FUNCTION_BLOCK FB_PackML_ExternalControl IMPLEMENTS ITF_PackML_ExternalControl
VAR_INPUT
END_VAR
VAR_OUTPUT
END_VAR
VAR
	nMode				: DINT;
	nModeCommand		: DINT;
	bModeCommandPulse	: BOOL;
	eState				: Tc3_PackML_V2.E_PMLState;
	eStateCommand		: Tc3_PackML_V2.E_PMLCommand;
	bStateCommandPulse	: BOOL;
	
	bStartPressed		: BOOL;
	bStartEnabled		: BOOL;
	bStopPressed		: BOOL;
	bStopEnabled		: BOOL;
	bResetPressed		: BOOL;
	bResetEnabled		: BOOL;
	bClearPressed		: BOOL;
	bClearEnabled		: BOOL;	
	
END_VAR

//Handle button presses
IF bStartPressed THEN
	IF eState = Tc3_PackML_V2.E_PMLState.ePMLState_Idle THEN
		eStateCommand := Tc3_PackML_V2.E_PMLCommand.ePMLCommand_Start;
		bStateCommandPulse := TRUE;
	ELSIF eState = Tc3_PackML_V2.E_PMLState.ePMLState_Held THEN
		eStateCommand := Tc3_PackML_V2.E_PMLCommand.ePMLCommand_Unhold;
		bStateCommandPulse := TRUE;
	END_IF
	bStartPressed := FALSE;
END_IF

IF bStopPressed THEN
	eStateCommand := Tc3_PackML_V2.E_PMLCommand.ePMLCommand_Stop;
	bStateCommandPulse := TRUE;
	bStopPressed := FALSE;
END_IF

IF bResetPressed THEN
	eStateCommand := Tc3_PackML_V2.E_PMLCommand.ePMLCommand_Reset;
	bStateCommandPulse := TRUE;
	bResetPressed := FALSE;
END_IF

IF bClearPressed THEN
	eStateCommand := Tc3_PackML_V2.E_PMLCommand.ePMLCommand_Clear;
	bStateCommandPulse := TRUE;
	bClearPressed := FALSE;
END_IF

//Handle enabling of the Start button
IF 		eState = Tc3_PackML_V2.E_PMLState.ePMLState_Idle
	OR	eState = Tc3_PackML_V2.E_PMLState.ePMLState_Held 	THEN
	bStartEnabled := TRUE;
ELSE
	bStartEnabled := FALSE;
END_IF

//Handle enabling of the Stop button
IF 		eState <> Tc3_PackML_V2.E_PMLState.ePMLState_Stopped
	AND	eState <> Tc3_PackML_V2.E_PMLState.ePMLState_Clearing
	AND	eState <> Tc3_PackML_V2.E_PMLState.ePMLState_Aborted
	AND	eState <> Tc3_PackML_V2.E_PMLState.ePMLState_Aborting
	AND	eState <> Tc3_PackML_V2.E_PMLState.ePMLState_Undefined 	THEN
	bStopEnabled := TRUE;
ELSE
	bStopEnabled := FALSE;
END_IF

//Handle enabling of the Reset button
IF 		eState = Tc3_PackML_V2.E_PMLState.ePMLState_Complete
	OR	eState = Tc3_PackML_V2.E_PMLState.ePMLState_Stopped 	THEN
	bResetEnabled := TRUE;
ELSE
	bResetEnabled := FALSE;
END_IF

//Handle enabling of the Clear button
IF 		eState = Tc3_PackML_V2.E_PMLState.ePMLState_Aborted	THEN
	bClearEnabled := TRUE;
ELSE
	bClearEnabled := FALSE;
END_IF


// Handle mode changes


PROPERTY ClearEnabled : BOOL
GET
ClearEnabled := bClearEnabled;
END_GET
SET
bClearEnabled := ClearEnabled;
END_SET
END_PROPERTY


PROPERTY ClearPressed : BOOL
GET
ClearPressed := bClearPressed;
END_GET
SET
bClearPressed := ClearPressed;
END_SET
END_PROPERTY

PROPERTY Mode : DINT
GET
Mode := nMode;
END_GET
SET
nMode := Mode;
END_SET
END_PROPERTY


PROPERTY ModeCommand : DINT
GET
ModeCommand := nModeCommand;
END_GET
SET
nModeCommand := ModeCommand;
END_SET
END_PROPERTY


PROPERTY ModeCommandPulse : BOOL
GET
ModeCommandPulse := bModeCommandPulse;
END_GET
SET
bModeCommandPulse := ModeCommandPulse;
END_SET
END_PROPERTY


PROPERTY ResetEnabled : BOOL
GET
ResetEnabled := bResetEnabled;
END_GET
SET
bResetEnabled := ResetEnabled;
END_SET
END_PROPERTY


PROPERTY ResetPressed : BOOL
GET
bResetPressed := ResetPressed;
END_GET
SET
bResetPressed := ResetPressed;
END_SET
END_PROPERTY


PROPERTY StartEnabled : BOOL
GET
StartEnabled := bStartEnabled;
END_GET
SET
bStartEnabled := StartEnabled;
END_SET
END_PROPERTY


PROPERTY StartPressed : BOOL
GET
StartPressed := bStartPressed;
END_GET
SET
bStartPressed := StartPressed;
END_SET
END_PROPERTY


PROPERTY State : Tc3_PackML_V2.E_PMLState
GET
State := eState;
END_GET
SET
eState := State;
END_SET
END_PROPERTY


PROPERTY StateCommand : Tc3_PackML_V2.E_PMLCommand
GET
StateCommand := eStateCommand;
END_GET
SET
eStateCommand := StateCommand;
END_SET
END_PROPERTY


PROPERTY StateCommandPulse : BOOL
GET
StateCommandPulse := bStateCommandPulse;
END_GET
SET
bStateCommandPulse := StateCommandPulse;
END_SET
END_PROPERTY


PROPERTY StopEnabled : BOOL
GET
StopEnabled := bStopEnabled;
END_GET
SET
bStopEnabled := StopEnabled;
END_SET
END_PROPERTY


PROPERTY StopPressed : BOOL
GET
StopPressed := bStopPressed;
END_GET
SET
bStopPressed := StopPressed;
END_SET
END_PROPERTY

END_FUNCTION_BLOCK

(* stored: Version 1.1.0.1, ProductVersion 3.1.4024.9
   POU FB_PackML_ExternalControl: Id {c53e3943-5b98-43e1-bdc9-fc1cc29d42fb}, SpecialFunc None
   Folder Simplified: Id {cd350b67-3bc4-40d9-a48c-43ed2012eac9}
   Folder Standard: Id {0ffae47d-ff66-4206-9cc7-d82722063454}
   Property ClearEnabled: Id {f86cd3a3-84af-4278-b7bc-9f3f839062c6}
   Get Get: Id {6a82a337-dc62-4320-bc89-97d7ecfe5261}
   Set Set: Id {6e97bad8-d173-4969-9a92-8b646746bb7f}
   Property ClearPressed: Id {4dab9de2-6548-4410-acc4-85210ecda5a6}
   Get Get: Id {a88997df-989c-46b0-805b-9476e4b5efed}
   Set Set: Id {efc5b417-03af-4b4d-a5a8-c0adf6759c1d}
   Property Mode: Id {c7ea0e58-ca4e-4e99-b638-fe78166e876e}
   Get Get: Id {70218e88-64c8-4f63-8a80-acfd4045de84}
   Set Set: Id {13511cb8-ed13-480c-86ff-84f7f4659e15}
   Property ModeCommand: Id {c1db968a-9663-400b-8205-1cfeb66a7c69}
   Get Get: Id {31c32bd1-9c86-4c24-bf49-81ec6a7d4c0f}
   Set Set: Id {9921b3f6-be46-4801-8dd5-2efe42107494}
   Property ModeCommandPulse: Id {9fcb23dd-067c-4e96-976c-d43f0d87af5b}
   Get Get: Id {5b9f0547-43d1-457b-85a4-545eb5c84dcd}
   Set Set: Id {b325549a-9de6-4caf-b9a1-c1dd2d13e760}
   Property ResetEnabled: Id {6c884262-09f4-4397-a880-f98840e975c5}
   Get Get: Id {e81768fd-c8d0-4323-ae4f-1c9cf5e166db}
   Set Set: Id {2a51cb31-3e56-4460-afe2-8cc0ebbd199d}
   Property ResetPressed: Id {9a66fef4-410e-49dd-99d0-530cf11460ec}
   Get Get: Id {b0dc1317-9ab3-43f7-9513-845d72a404d9}
   Set Set: Id {877bb0df-6f2b-4eb2-b4b0-5e68d95eb78e}
   Property StartEnabled: Id {c34d85d1-e716-4911-8cc6-928f8c00f703}
   Get Get: Id {69b3a00c-e55b-47ee-9ae6-55c7e9288b22}
   Set Set: Id {f3d5b72d-e4a9-4071-91e3-b6796c260079}
   Property StartPressed: Id {1b95041d-a087-4acb-8cee-7190cb3dd908}
   Get Get: Id {c9e4cc9d-fa48-4bd2-9585-23378d4b7a92}
   Set Set: Id {1291f257-39ed-45e5-b2c2-dbf77f6d95df}
   Property State: Id {6642fb50-7898-43b1-935b-c91ff6dd5a87}
   Get Get: Id {ba3baffa-8421-4fea-b76c-68697f856880}
   Set Set: Id {43212634-bcea-481a-b525-7feb8c999f70}
   Property StateCommand: Id {1eb71234-fc01-4c3d-8f9e-a869a63098e6}
   Get Get: Id {0ad453dc-9a75-4fff-9e3c-26351eda763a}
   Set Set: Id {42b65406-59b0-4ee4-bd33-c6de0bc2bf37}
   Property StateCommandPulse: Id {ca898e5e-196d-43bb-b5db-9bca6560c220}
   Get Get: Id {98df8afe-3734-4bea-95fa-f67aedf46299}
   Set Set: Id {6c12848f-eb01-4f74-b223-322e4a4d403d}
   Property StopEnabled: Id {73c73278-a15a-48d1-9e83-45efc93f4db9}
   Get Get: Id {2fd959fa-0ebb-4238-9f60-89a2e43a75c7}
   Set Set: Id {6b4a205f-d47e-41fc-87d4-a1667d2995b0}
   Property StopPressed: Id {e906d0fc-e1f1-4dd7-bab3-3850b481fd23}
   Get Get: Id {1456d948-cc82-4c0f-889d-3e970105ab22}
   Set Set: Id {bb3cb8ac-06c8-41d8-b6cb-0a818f1c34f0} *)
